// TIA Portal V20 export
DATA_BLOCK "SBK08"   // DB212
// stored: MemoryReserve 100
   VAR
      "X1-0 Gate EC RH: Lock" : Bool;
      "X2-1 Gate EC RH: Reset" : Bool;
      "X3-2 reserved" : Bool;
      "X4-3 reserved" : Bool;
      "X1-4 Gate EC RH: Unlock" : Bool;
      "X2-5 reserved" : Bool;
      "X3-6 reserved" : Bool;
      "X4-7 reserved" : Bool;
      "X5-0 Gate EC RH: Lock lamp on" : Bool;
      "X6-1 Gate EC RH: Unlock lamp on" : Bool;
      "X7-2 Gate EC RH: Reset lamp on" : Bool;
   END_VAR
BEGIN
END_DATA_BLOCK
